{attribute 'GeneratedUsingTerminal: EL4102--0000'}
{attribute addProperty BoxType "EL4102--0000"}
{attribute addProperty Id "OutputAT %Q*INT2"}
{attribute addProperty CRC "1604026022"}
{attribute addProperty Size "2"}
TYPE Channel_5F9B7EA6 :
STRUCT
	{attribute addProperty Name "Output"}
	Output AT %Q* : INT;
END_STRUCT
END_TYPE

(* stored: Version 1.2.0.0, ProductVersion 3.1.4024.9
   DUT Channel_5F9B7EA6: Id {bc92924f-953a-454c-9b03-7c215ed82bbf} *)
